TYPE MyExampleStructure :
STRUCT
	myInt : INT := 123;
	myBool : BOOL := TRUE;
	myString : STRING := 'hello';
	myArray : ARRAY[0..1] OF BYTE := [0, 255];
	myInternalStructure : MyExampleInternalStructure;
END_STRUCT
END_TYPE

(* stored: Version 1.1.0.1, ProductVersion 3.1.4024.12
   DUT MyExampleStructure: Id {d4c564c2-b74d-4b48-9d3d-7316d9cf8f4f} *)
